(*
SPDX-FileCopyrightText: © 2026 Oleksandr Tiutyk <trofimich@gmail.com>
SPDX-License-Identifier: MIT
License: https://opensource.org/license/mit
*)

{attribute 'no_explicit_call' := 'do not call this function block directly'} 
PROGRAM SystemAnyTypes
VAR
	{attribute 'hide'} 
	_ClassName : STRING := __POUNAME();
END_VAR

METHOD CheckIsNull : BOOL
VAR_INPUT
	value : __SYSTEM.AnyType;
END_VAR
CheckIsNull := value.pValue = 0 OR_ELSE value.diSize = 0 OR_ELSE value.TypeClass = __SYSTEM.TYPE_CLASS.TYPE_NONE;
END_METHOD

{attribute 'monitoring' := 'call'}
PROPERTY ClassName : REFERENCE TO STRING
GET
ClassName REF= _ClassName;
END_GET
END_PROPERTY

METHOD CreateAnyTypeByAny : __SYSTEM.AnyType
VAR_INPUT
	anyValue : ANY;
END_VAR
CreateAnyTypeByAny := anyValue;
END_METHOD

METHOD CreateAnyTypeByGenericValue : __SYSTEM.AnyType
VAR_IN_OUT CONSTANT
	genericValue : GENERIC_VALUE;
END_VAR
CreateAnyTypeByGenericValue.TypeClass := SystemTypeClassConvertor.GetSystemTypeClassByGenericTypeClass(genericValue.TypeClass);
CreateAnyTypeByGenericValue.pValue := genericValue.Address;
CreateAnyTypeByGenericValue.diSize := TO_DINT(genericValue.Size);
END_METHOD

{attribute 'monitoring' := 'call'}
PROPERTY NamespaceName : REFERENCE TO STRING
GET
NamespaceName REF= CurrentNamespace.Name;
END_GET
END_PROPERTY

END_PROGRAM

(* stored: Version 1.1.0.1
   POU SystemAnyTypes: Id {6a7e7caf-8e80-4ccf-abb4-b450c8a2b399}, SpecialFunc None
   Method CheckIsNull: Id {6872bbfd-fcf4-4ff1-8861-988ed289e280}
   Property ClassName: Id {bc62ea28-f530-4c6b-8182-b79f5d9e4fc4}
   Get Get: Id {77144c18-f2c0-4f0f-bd6d-c1cae1fcd65a}
   Method CreateAnyTypeByAny: Id {1f2becd5-4a43-4d75-827f-7c56c084215c}
   Method CreateAnyTypeByGenericValue: Id {73f9d3c1-a03b-4864-9d65-f396047544c5}
   Property NamespaceName: Id {8304df90-847d-4024-9242-86baaf0a63ef}
   Get Get: Id {847b0818-cabd-4275-a44e-d5ee2eb75ef9} *)
